INTERFACE PUBLIC SuspendingCommands EXTENDS RunningStateCommands, ActionStateCommands, HoldableStateCommands

END_INTERFACE

(* stored: Version 1.1.0.1, ProductVersion 3.1.4026.18
   Itf SuspendingCommands: Id {293f49ed-8bfe-09e2-1376-339448adb778} *)
